Staubli VAL3: sCenterRow.pgx

program sCenterRow(string& x_sRow)
begin

  //max length 40 characters
  call sCenterString(x_sRow,asc(" ",0),40)

end
